// TIA Portal V17 export
// export: Created 2025-03-05T08:02:17.5706413Z, ExportSetting WithDefaults, DisplayName Totally Integrated Automation Portal, DisplayVersion V17 Update 8, DisplayName TIA Portal Openness, DisplayVersion V17 Update 8, DisplayName TIA Portal Version Control Interface, DisplayVersion V17, DisplayName SINAMICS Startdrive Advanced, DisplayVersion V17 SP2, DisplayName SINAMICS Startdrive G110M, G120, G120C, G120D, G120P, G115D, DisplayVersion V17 SP2, DisplayName SINAMICS Startdrive G130, G150, S120, S150, SINAMICS MV, S210, DisplayVersion V17 SP2, DisplayName STEP 7 Professional, DisplayVersion V17 Update 8, DisplayName SINUMERIK ONE STEP 7 Toolbox, DisplayVersion V17 Update 12, DisplayName SINUMERIK 840D sl STEP 7 Toolbox, DisplayVersion V17 Update 12, DisplayName STEP 7 Safety, DisplayVersion V17 Update 6, DisplayName WinCC Advanced, DisplayVersion V17 Update 8
TYPE "DIAGNOSTIC_MOD"
// stored: IsFailsafeCompliant false
   STRUCT
      CHANNEL_1_STATE : Bool;   // CHANNEL 1 STATE
      CHANNEL_2_STATE : Bool;   // CHANNEL 2 STATE
      CHANNEL_3_STATE : Bool;   // CHANNEL 3 STATE
      CHANNEL_4_STATE : Bool;   // CHANNEL 4 STATE
      CHANNEL_1_ALARM : Bool;   // CHANNEL 1 ALARM
      CHANNEL_2_ALARM : Bool;   // CHANNEL 2 ALARM
      CHANNEL_3_ALARM : Bool;   // CHANNEL 3 ALARM
      CHANNEL_4_ALARM : Bool;   // CHANNEL 4 ALARM
      MOD_ERROR_ALARM : Bool;   // MOD ERROR ALARM
   END_STRUCT;
END_TYPE
